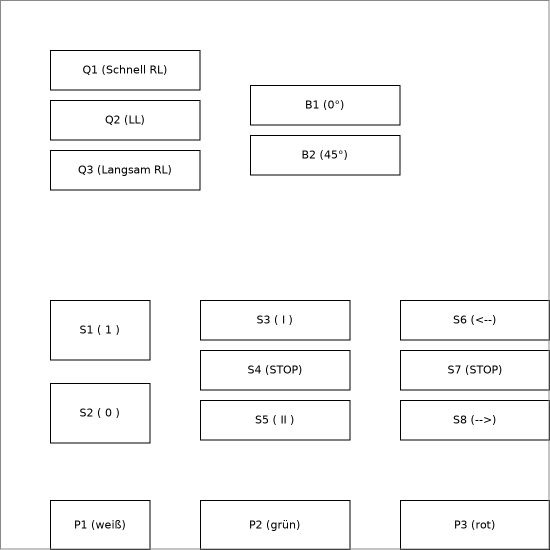
VISUALIZATION VisuGetriebemotor  // 550x550
    Rectangle (50,500 100x50), "P1 (weiß)", colour toggle: SimDA.P1
        tap SimDA.P1
    Rectangle (50,300 100x60), "S1 ( 1 )", colour toggle: SimDI.S1
    Rectangle (200,500 150x50), "P2 (grün)"
        tap SimDA.P2
    Rectangle (400,500 150x50), "P3 (rot)"
        tap SimDA.P3
    Rectangle (50,383 100x60), "S2 ( 0 )", colour toggle: SimDI.S2
    Rectangle (200,300 150x40), "S3 ( I )", colour toggle: SimDI.S3
    Rectangle (200,350 150x40), "S4 (STOP)", colour toggle: SimDI.S4
    Rectangle (200,400 150x40), "S5 ( II )", colour toggle: SimDI.S5
    Rectangle (400,300 150x40), "S6 (<--)", colour toggle: SimDI.S6
    Rectangle (400,350 150x40), "S7 (STOP)", colour toggle: SimDI.S7
    Rectangle (400,400 150x40), "S8 (-->)", colour toggle: SimDI.S8
    Rectangle (50,50 150x40), "Q1 (Schnell RL)"
        tap SimDA.Q1
    Rectangle (50,100 150x40), "Q2 (LL)"
        tap SimDA.Q2
    Rectangle (50,150 150x40), "Q3 (Langsam RL)"
        tap SimDA.Q3
    Rectangle (250,85 150x40), "B1 (0°)", colour toggle: SimDI.B1
    Rectangle (250,135 150x40), "B2 (45°)", colour toggle: SimDI.B2
END_VISUALIZATION

(* stored: Version 1.1.0.1, ProductVersion 3.1.4024.5
   Visu VisuGetriebemotor: Id {f31a0e65-aa70-4d08-b440-27b2419b6551} *)
